// TIA Portal V16 export
// export: Created 2023-08-28T09:37:30.4698976Z, ExportSetting WithDefaults, DisplayName Totally Integrated Automation Portal, DisplayVersion V16 Update 6, DisplayName TIA Portal Version Control Interface, DisplayVersion V16 Update 2, DisplayName TIA Portal Openness, DisplayVersion V16 Update 6, DisplayName STEP 7 Professional, DisplayVersion V16 Update 6, DisplayName STEP 7 Safety, DisplayVersion V16, DisplayName WinCC Advanced, DisplayVersion V16 Update 6
FUNCTION_BLOCK "00_S_WatchDog PLC - WinCC"   // FB13, LAD
TITLE = WatchDog PLC - WinCC
{ S7_Optimized_Access := 'TRUE' }
AUTHOR : rtecmer
VERSION : 0.1
// Kontrola komunikacji PLC z WinCC SCADA . Zerwanie komunikacji przekazywane do WinCC SCADA i PLC Master S7-300 (RS3)
// stored: AutoNumber true, IsIECCheckEnabled false, IsRetainMemResEnabled false, MemoryReserve 500, SetENOAutomatically false, UDAEnableTagReadback false
   VAR_TEMP   // added for the SCL form of the ladder/FBD networks
      _w1 : Bool;
      _w2 : Bool;
   END_VAR
BEGIN

REGION Network 1: WatchDog WinCC - PLC
   // Konfiguracja WinCC Flexible - ustawiony Area Point (Coordination) na DB29 DBW12
   // WinCC wpisuje z częstotliwością 0,9s na zmianę wartości 1 i 5.
   // PLC  kontroluje tę zmianę poprzez Timer TON z histerezą 10s. Jeśli nastąpi przerwanie komunikacji
   // zasygnalizuje to jeden z dwóch TON ustawiając możliwość inkrementacji zmiennej pomocniczej w instancji "Dane_ComunicationControlHMI".tempWatchDog_WinCC i ustawi bitu alarmu braku komunikacji z WinCC  
   // Po powrocie komunikacji zmienna "Dane_ComunicationControlHMI".tempWatchDog_WinCC jest zerowana.
   // Wartośc zmiennej  "Dane_ComunicationControlHMI".tempWatchDog_WinCC jest pobierana przez scipt VB WinCC jeśli jest 0 to comunikacja OK jeśli natomiast  > 0 to script VB inkrementuje wewnętrzną zmienną i ustawia alarm w WinCC.
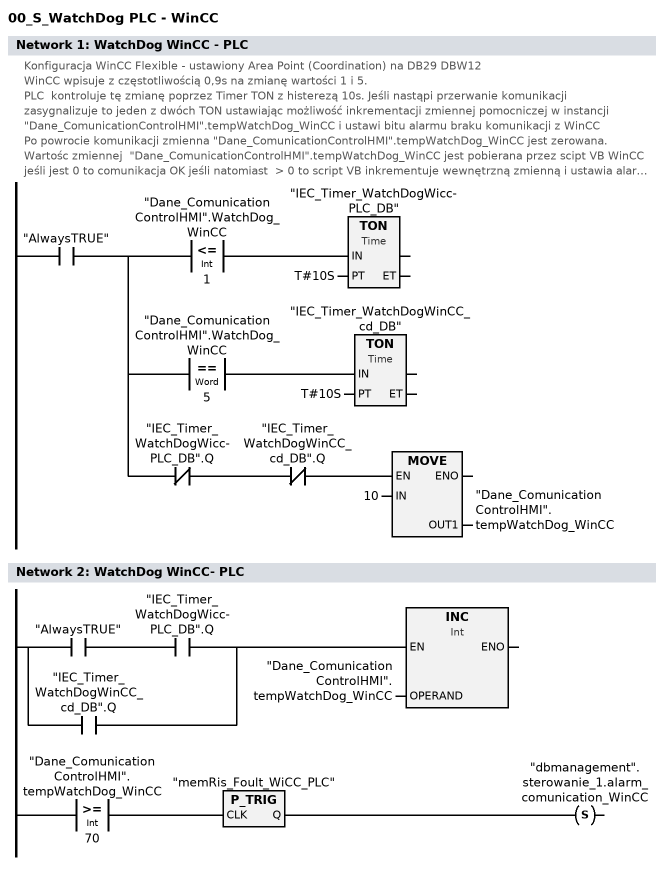
   RUNG wire#powerrail
      Contact( "AlwaysTRUE" )
      wire#w1
      { S7_Templates := "SrcType := Int" } LE_Contact(in1 := "Dane_ComunicationControlHMI".WatchDog_WinCC, in2 := 1)
      { S7_Templates := "time_type := Time" } "IEC_Timer_WatchDogWicc-PLC_DB".TON(pt := T#10S, et =>)
   END_RUNG
   RUNG wire#w1
      { S7_Templates := "SrcType := Word" } EQ_Contact(in1 := "Dane_ComunicationControlHMI".WatchDog_WinCC, in2 := 5)
      { S7_Templates := "time_type := Time" } "IEC_Timer_WatchDogWinCC_cd_DB".TON(pt := T#10S, et =>)
   END_RUNG
   RUNG wire#w1
      I_Contact( "IEC_Timer_WatchDogWicc-PLC_DB".Q )
      I_Contact( "IEC_Timer_WatchDogWinCC_cd_DB".Q )
      Move(in := 10, out1 => "Dane_ComunicationControlHMI".tempWatchDog_WinCC)
   END_RUNG
   // the same network as SCL:
   "IEC_Timer_WatchDogWicc-PLC_DB".TON(IN := "AlwaysTRUE" AND ("Dane_ComunicationControlHMI".WatchDog_WinCC <= 1),
                           PT := T#10S);
   "IEC_Timer_WatchDogWinCC_cd_DB".TON(IN := "AlwaysTRUE" AND ("Dane_ComunicationControlHMI".WatchDog_WinCC = 5),
                           PT := T#10S);
   IF "AlwaysTRUE" AND NOT "IEC_Timer_WatchDogWicc-PLC_DB".Q AND NOT "IEC_Timer_WatchDogWinCC_cd_DB".Q THEN
       "Dane_ComunicationControlHMI".tempWatchDog_WinCC := 10;
   END_IF;
END_REGION

REGION Network 2: WatchDog WinCC- PLC
   RUNG wire#powerrail
      Contact( "AlwaysTRUE" )
      Contact( "IEC_Timer_WatchDogWicc-PLC_DB".Q )
      wire#w1
      { S7_Templates := "DestType := Int" } Inc( "Dane_ComunicationControlHMI".tempWatchDog_WinCC )
   END_RUNG
   RUNG wire#powerrail
      Contact( "IEC_Timer_WatchDogWinCC_cd_DB".Q )
   END_RUNG wire#w1
   RUNG wire#powerrail
      { S7_Templates := "SrcType := Int" } GE_Contact(in1 := "Dane_ComunicationControlHMI".tempWatchDog_WinCC, in2 := 70)
      P_Trig( "memRis_Foult_WiCC_PLC" )
      S_Coil( "dbmanagement".sterowanie_1.alarm_comunication_WinCC )
   END_RUNG
   // the same network as SCL:
   IF ("AlwaysTRUE" AND "IEC_Timer_WatchDogWicc-PLC_DB".Q) OR "IEC_Timer_WatchDogWinCC_cd_DB".Q THEN
       "Dane_ComunicationControlHMI".tempWatchDog_WinCC := "Dane_ComunicationControlHMI".tempWatchDog_WinCC + 1;
   END_IF;
   #_w1 := "Dane_ComunicationControlHMI".tempWatchDog_WinCC >= 70;
   #_w2 := #_w1 AND NOT "memRis_Foult_WiCC_PLC";   // rising edge
   "memRis_Foult_WiCC_PLC" := #_w1;
   IF #_w2 THEN "dbmanagement".sterowanie_1.alarm_comunication_WinCC := TRUE; END_IF;
END_REGION
END_FUNCTION_BLOCK
